TYPE TcoRotaryTransfer_Control EXTENDS TcoCore.TcoStruct:
STRUCT

	
		
END_STRUCT
END_TYPE

(* stored: Version 1.1.0.1
   DUT TcoRotaryTransfer_Control: Id {f17d4c1d-7b6b-4c09-99d2-70695cdd83bc} *)
